// TwinCAT 3 PLC project ToolChanger
// ProgramVersion: 3.1.4023.0
// libraries:
//   CmpBitmapPool, * (System)
//   Tc2_MC2, * (Beckhoff Automation GmbH)
//   Tc2_NC, * (Beckhoff Automation GmbH)
//   Tc2_Standard, * (Beckhoff Automation GmbH)
//   Tc2_System, * (Beckhoff Automation GmbH)
//   Tc2_Utilities, * (Beckhoff Automation GmbH)
//   Tc3_Module, * (Beckhoff Automation GmbH)
//   VisuDialogs, * (System)
//   VisuSymbols,3.5.10.0,System
// project tree:
//   / GlobalTextList.TcGTLO, PlcTask.TcTTO, Visualization Manager.TcVMO (not stored)
//   GVLs/ Allengage.TcGVL, CLEANout.TcGVL, cntrlstate.TcGVL, DSin.TcGVL, DSout.TcGVL, engage.TcGVL, TCin.TcGVL, TCout.TcGVL
//   POUs/FBs/Cleaner/ fb_cleanIn.TcPOU, fb_cleanOut.TcPOU
//   POUs/FBs/Combined/ fb_engageDockAll.TcPOU, fb_engageUndockAll.TcPOU
//   POUs/FBs/DS/ fb_dsopenclose.TcPOU
//   POUs/FBs/Safety/ fb_NozCheck.TcPOU, fb_switchclkcheck.TcPOU
//   POUs/FBs/TC/ fb_dock.TcPOU, fb_toggleVal.TcPOU, fb_undock.TcPOU
//   POUs/FBs/Testing/ fb_testpiston.TcPOU
//   POUs/ MAIN.TcPOU
//   VISUs/ ImagePool.TcIPO (not stored), Visualization.TcVIS
// real-time tasks:
//   TASK PlcTask: cycle T#10ms, priority 20, ADS port 350
// motion (NC):
//   TASK NC-Task 1 SAF: cycle T#2ms, priority 4, ADS port 501
//   TASK NC-Task 1 SVB: cycle T#10ms, priority 8, ADS port 511
//   AXIS Axis 1 (id 1)
//     Velo: SlowManual=20, FastManual=20
//     OtherSettings: AllowMotionCmdToSlave=true
//     encoder EncType=1
//     drive DrvType=5
//       Analog: TorqueSetpointScale=10, ScaleFactorActTorque=0.1
//       TimeComp: TaskDelayCycles=1
//     controller CtrType=1
//       CtrPara: PriorControlFactor=1
//         Observer: BandWidth=20
// I/O:
//   DEVICE Device 1 (EtherCAT), AmsNetId 192.168.1.12.2.1
//     Term 1 (EK1200) [EK1200-5000 EtherCAT Power supply (2A E-Bus)]
//       Term 2 (EL1008) [EL1008 8Ch. Dig. Input 24V, 3ms]
//       Term 3 (EL2008) [EL2008 8Ch. Dig. Output 24V, 0.5A]
//       Term 4 (EK1110) [EK1110 EtherCAT extension]
//   DEVICE Device 4 (COM Port)
// variable links:
//   ToolChanger/ToolChanger Instance <-> Device 1 (EtherCAT)/Term 1 (EK1200)/Term 2 (EL1008)
//     PlcTask Inputs/DSin.endStopBck <-> Channel 5/Input
//     PlcTask Inputs/DSin.endStopFrnt <-> Channel 4/Input
//     PlcTask Inputs/TCin.CollisionSW <-> Channel 2/Input
//     PlcTask Inputs/TCin.ProxDwn <-> Channel 1/Input
//     PlcTask Inputs/TCin.ProxUp <-> Channel 3/Input
//   ToolChanger/ToolChanger Instance <-> Device 1 (EtherCAT)/Term 1 (EK1200)/Term 3 (EL2008)
//     PlcTask Outputs/DSout.servoBackward <-> Channel 4/Output
//     PlcTask Outputs/DSout.servoForward <-> Channel 2/Output
//     PlcTask Outputs/TCout.valvepull <-> Channel 1/Output
//     PlcTask Outputs/TCout.valvepush <-> Channel 3/Output
//   ToolChanger/ToolChanger Instance <-> NC-Task 1 SAF/Axes/Axis 1
//     PlcTask Inputs/MAIN.opcl.ax1.NcToPlc <-> Outputs/ToPlc
//     PlcTask Outputs/MAIN.opcl.ax1.PlcToNc <-> Inputs/FromPlc

CONFIGURATION ToolChanger
    RESOURCE PLC ON TwinCAT3
        TASK PlcTask(INTERVAL := T#10ms, PRIORITY := 20);
        PROGRAM MAIN WITH PlcTask : MAIN;
    END_RESOURCE
END_CONFIGURATION

// ---- GVLs/Allengage.TcGVL
{attribute 'qualified_only'}
VAR_GLOBAL
	cleanInd: BOOL := FALSE;
	cleanOutd: BOOL := FALSE;
	cleanInu: BOOL := FALSE;
	cleanOutu: BOOL := FALSE;
	undock: BOOL := FALSE;
	dock: BOOL := FALSE;
	stepopen: BOOL := FALSE;
	stepclose: BOOL := FALSE;
	stepper : BOOL := FALSE;
END_VAR

// ---- GVLs/CLEANout.TcGVL
{attribute 'qualified_only'}
VAR_GLOBAL
	// Inside cleaner valve
	inValve AT %Q*: BOOL;
	// Outside cleaner valve
	outValve AT %Q*: BOOL;
	
	// ADD COVER SERVO TO SOLUTION
END_VAR

// ---- GVLs/cntrlstate.TcGVL
{attribute 'qualified_only'}
VAR_GLOBAL
	undock: BOOL;
	dock: BOOL;
	cleanin: BOOL;
	cleanout: BOOL;
	piston_moving: BOOL;
	cover_moving: BOOL;
END_VAR

// ---- GVLs/DSin.TcGVL
{attribute 'qualified_only'}
VAR_GLOBAL
	// Cover switch back
	endStopBck AT %I*: BOOL;
	// Cover switch front
	endStopFrnt AT %I*: BOOL;
	// stepper engagement
	open : BOOL := FALSE;
	close : BOOL := FALSE;
	ID: INT;
END_VAR

// ---- GVLs/DSout.TcGVL
{attribute 'qualified_only'}
VAR_GLOBAL
	//ADD COVER SERVO AND STEPPER MOTOR TO SOLUTION
	servoBackward AT %Q*: BOOL := FALSE;
	servoForward AT %Q*: BOOL := false;
END_VAR

// ---- GVLs/engage.TcGVL
{attribute 'qualified_only'}
VAR_GLOBAL
	cleanIn: BOOL := FALSE;
	cleanOut: BOOL := FALSE;
	undock: BOOL := FALSE;
	dock: BOOL := FALSE;
	stepopen: BOOL := FALSE;
	stepclose: BOOL := FALSE;
	stepper : BOOL := FALSE;
	allundock: BOOL :=FALSE;
	alldock: BOOL :=FALSE;
	pisttest : BOOL := FALSE;
END_VAR

// ---- GVLs/TCin.TcGVL
{attribute 'qualified_only'}
VAR_GLOBAL
	// Upper inductive sensor
	ProxUp AT %I*: BOOL;
	// Lower inductive sensor
	ProxDwn AT %I*: BOOL;
	// Safety limit switch
	CollisionSW AT %I*: BOOL;
	// Most significant bit
	ID1 AT %I*: BOOL := TRUE;
	// Middle bit
	ID2 AT %I*: BOOL;
	// Least significant bit
	ID3 AT %I*: BOOL;
	toolOn : BOOL;
END_VAR

// ---- GVLs/TCout.TcGVL
{attribute 'qualified_only'}
VAR_GLOBAL
	// Dual valve control
	valvepush AT %Q*: BOOL := TRUE;
	valvepull AT %Q*: BOOL;
	// Limit switch clock signal
	SwCLK AT %Q*: BOOL;
END_VAR

// ---- POUs/MAIN.TcPOU
PROGRAM MAIN
VAR
	cleanin: fb_cleanIn;
	cleanout: fb_cleanOut;
	undock: fb_undock;
	dock: fb_dock;
	switchclk: fb_switchclkcheck;
	opcl: fb_dsopenclose;
	allundock: fb_engageUndockAll;
	alldock: fb_engageDockAll;
	stop : TC_Stop;
	pisttest: fb_testpiston;
END_VAR

(*always running*)

IF TCin.toolOn THEN
	switchclk();
END_IF

(*engaged manually*)
IF engage.stepper THEN
	opcl();
END_IF

IF engage.cleanIn THEN
	cntrlstate.cleanin := FALSE;
	cleanin(done := cntrlstate.cleanin);
	IF cntrlstate.cleanin THEN
		engage.cleanIn := FALSE;
	END_IF
END_IF

IF engage.cleanOut THEN
	cntrlstate.cleanout := FALSE;
	cleanout(done := cntrlstate.cleanout);
	IF cntrlstate.cleanout THEN
		engage.cleanOut := FALSE;
	END_IF
END_IF

IF engage.undock THEN
	cntrlstate.undock := FALSE;
	undock();
	IF cntrlstate.undock THEN
		engage.undock := FALSE;
	END_IF
END_IF

IF engage.dock THEN
	cntrlstate.dock := FALSE;
	dock(toolID := 4);
	IF cntrlstate.dock THEN
		engage.dock := FALSE;
	END_IF
END_IF


(*engage a sequence*)
IF engage.allundock THEN
	allundock();
END_IF

IF engage.alldock THEN
	alldock();
END_IF

(*errorHandle stopping plc*)
IF NOT switchclk.swXgood THEN
	stop(STOP:=TRUE);
END_IF


(*TESTING*)
IF engage.pisttest THEN
	pisttest();
END_IF

END_PROGRAM

// ---- POUs/FBs/Cleaner/fb_cleanIn.TcPOU
FUNCTION_BLOCK fb_cleanIn
VAR_INPUT
	IN: BOOL;
END_VAR
VAR_OUTPUT
END_VAR
VAR
	wait: TON;
	step: INT;
END_VAR

VAR_IN_OUT
	done: BOOL;
END_VAR

CASE step OF
	0:
		IF NOT done THEN
			cleanout.inValve := TRUE;
			wait(IN := TRUE, PT := T#5S);
			step := 1;
		END_IF
	1:
		IF wait.Q THEN
			wait.IN := FALSE;
			cleanout.inValve := FALSE;
			step := 2;
		END_IF
		
	2: 
		step := 0;
		done := TRUE;
	
END_CASE
wait();

END_FUNCTION_BLOCK

// ---- POUs/FBs/Cleaner/fb_cleanOut.TcPOU
FUNCTION_BLOCK fb_cleanOut
VAR_INPUT
END_VAR
VAR_OUTPUT
END_VAR
VAR
	step: INT;
	wait: TON;
END_VAR

VAR_IN_OUT
	done: BOOL;
END_VAR

CASE step OF
	0:
		IF NOT done THEN
			cleanout.outValve := TRUE;
			wait(IN := TRUE, PT := T#5S);
			step := 1;
		END_IF
	1:
		IF wait.Q THEN
			wait.IN := FALSE;
			cleanout.outValve := FALSE;
			step := 2;
		END_IF
		
	2: 
		step := 0;
		done := TRUE;
	
END_CASE
wait();

END_FUNCTION_BLOCK

// ---- POUs/FBs/TC/fb_undock.TcPOU
FUNCTION_BLOCK fb_undock
VAR_INPUT
END_VAR
VAR_OUTPUT
END_VAR
VAR
	step: INT;
	unLock: fb_toggleVal;
END_VAR

CASE step OF
	0:
		IF NOT tcin.ProxUp THEN
			unLock(IN:= TRUE);
			unLock.IN := FALSE;
			cntrlstate.piston_moving := TRUE;
			step := 1;
		END_IF
	1: 
		IF tcin.ProxUp AND tcin.ProxUp THEN
			 cntrlstate.undock := TRUE;
			 cntrlstate.piston_moving := FALSE;
			 step := 0;
		END_IF
	99:
		//ERROR HANDLING
END_CASE
unLock();
(*
CASE step OF
	0:
		IF tcin.ProxDwn THEN
			unLock(IN:= TRUE);
			unLock.IN := FALSE;
			cntrlstate.piston_moving := TRUE;
			step := 1;
		END_IF
	1: 
		IF tcin.ProxUp AND NOT tcin.ProxDwn THEN
			 cntrlstate.undock := TRUE;
			 cntrlstate.piston_moving := FALSE;
			 step := 0;
		END_IF
	99:
		//ERROR HANDLING
END_CASE
unLock();*)

END_FUNCTION_BLOCK

// ---- POUs/FBs/TC/fb_toggleVal.TcPOU
FUNCTION_BLOCK fb_toggleVal
VAR_INPUT
	IN: BOOL;
END_VAR
VAR_OUTPUT
END_VAR
VAR
END_VAR

IF IN = TRUE AND TCin.ProxUp THEN
	TCout.valvepush := TRUE;
	TCout.valvepull := FALSE;
ELSIF IN = TRUE AND not TCin.ProxUp THEN
	TCout.valvepull := TRUE;
	TCout.valvepush := FALSE;
END_IF

(*
IF IN = TRUE AND TCin.ProxUp THEN
	TCout.valve := FALSE;
ELSIF IN = TRUE AND TCin.ProxDwn THEN
	TCout.valve := TRUE;
END_IF*)

END_FUNCTION_BLOCK

// ---- POUs/FBs/TC/fb_dock.TcPOU
FUNCTION_BLOCK fb_dock
VAR_INPUT
	toolID: int;
END_VAR
VAR_OUTPUT
END_VAR
VAR
	step: INT;
	Lock: fb_toggleVal;
	IDcheck: fb_NozCheck;
END_VAR

CASE step OF
	0:
		IF tcin.ProxUp THEN
			Lock(IN:= TRUE);
			Lock.IN := FALSE;
			cntrlstate.piston_moving := TRUE;
			step := 1;
		END_IF
	1: 
		IF NOT tcin.ProxUp AND NOT tcin.ProxUp THEN
			IDcheck(inID := toolID);
			cntrlstate.piston_moving := FALSE;
			IF IDcheck.good THEN
				cntrlstate.dock := TRUE;
				step := 0;
			ELSIF NOT IDcheck.good THEN
				step := 99;
			END_IF
			
		END_IF
	99:
		//ERROR HANDLING
END_CASE

END_FUNCTION_BLOCK

// ---- POUs/FBs/Safety/fb_NozCheck.TcPOU
FUNCTION_BLOCK fb_NozCheck
VAR_INPUT
	inID: INT;
END_VAR
VAR_OUTPUT
	good: BOOL;
	done: BOOL;
END_VAR
VAR
	outID: INT;
END_VAR

// example (ID1 = 0, ID2 = 1, ID3 = 1)=011 => outID = 3
good := FALSE;
done := FALSE;
IF TCin.ID1 = FALSE AND TCin.ID2 = FALSE AND TCin.ID3 = FALSE THEN
	outID := 0;
ELSIF TCin.ID1 = FALSE AND TCin.ID2 = FALSE AND TCin.ID3 = TRUE THEN
	outID := 1;
ELSIF TCin.ID1 = FALSE AND TCin.ID2 = TRUE AND TCin.ID3 = FALSE THEN
	outID := 2;	
ELSIF TCin.ID1 = FALSE AND TCin.ID2 = TRUE AND TCin.ID3 = TRUE THEN
	outID := 3;
ELSIF TCin.ID1 = TRUE AND TCin.ID2 = FALSE AND TCin.ID3 = FALSE THEN
	outID := 4;
ELSIF TCin.ID1 = TRUE AND TCin.ID2 = FALSE AND TCin.ID3 = TRUE THEN
	outID := 5;	
ELSIF TCin.ID1 = TRUE AND TCin.ID2 = TRUE AND TCin.ID3 = FALSE THEN
	outID := 6;	
ELSIF TCin.ID1 = TRUE AND TCin.ID2 = TRUE AND TCin.ID3 = TRUE THEN
	outID := 7;	
END_IF

IF inID = outID THEN
	good := TRUE;
	done := TRUE;
ELSIF inID <> outID THEN
	good := FALSE;
	done := TRUE;
END_IF

END_FUNCTION_BLOCK

// ---- POUs/FBs/Safety/fb_switchclkcheck.TcPOU
FUNCTION_BLOCK fb_switchclkcheck
VAR_OUTPUT
	swXgood: BOOL := TRUE;
END_VAR
VAR
	prev_clk: BOOL;
END_VAR

(*This function block sends an alternating signal at a frequency of 100 Hz, and checks whether 
it has been altered from previous check*)

(*
TCout.SwCLK := NOT TCout.SwCLK;	
IF prev_clk = TCout.SwCLK THEN
	swXgood := FALSE;
ELSE 
	swXgood := TRUE;
END_IF
prev_clk := TCout.SwCLK; //only for testing => when doing physical setup => prev_clk := TCin.CollisionSW; 
*)

IF TCin.CollisionSW = FALSE THEN
	// STOP
END_IF

END_FUNCTION_BLOCK

// ---- POUs/FBs/DS/fb_dsopenclose.TcPOU
FUNCTION_BLOCK fb_dsopenclose
VAR_INPUT
END_VAR
VAR_OUTPUT
END_VAR
VAR
	ax1: AXIS_REF;
	McJog: MC_Jog;
	McPower: MC_Power;
	McReset: MC_Reset;
	McStop: MC_Stop;
	iState: INT;
END_VAR

(*McPower(Axis := ax1, Enable := TRUE, Enable_Positive := TRUE, Enable_Negative := TRUE);
McReset(Axis := ax1);
McJog(Axis := ax1);
CASE iState OF 
	0: 
		iState := 10;
	
	10:
		McReset(Axis:= ax1, Execute := TRUE);
		IF McReset.Done THEN
			iState := 20;
		ELSIF McReset.Error THEN
			iState := 999;
		END_IF
	
	20:
		IF McPower.Status THEN
			iState := 30;
		END_IF
		
	30:
		IF engage.stepopen OR DSin.open THEN
			cntrlstate.cover_moving := TRUE;
			McJog(Axis := ax1, JogForward := NOT DSin.endStopBck, Velocity := 20);
			IF DSin.endStopBck THEN
				cntrlstate.cover_moving := FALSE;
				engage.stepper := FALSE;
				engage.stepopen := FALSE;
				DSin.open := FALSE;
			END_IF
		ELSIF engage.stepclose OR DSin.close THEN
			cntrlstate.cover_moving := TRUE;
			McJog(Axis := ax1, JogBackwards := NOT DSin.endStopFrnt, Velocity := 20);
			IF DSin.endStopFrnt THEN
				cntrlstate.cover_moving := FALSE;
				engage.stepper := FALSE;
				engage.stepclose := FALSE;
				DSin.close := FALSE;
			END_IF
		END_IF
END_CASE
*)
IF engage.stepopen OR DSin.open THEN
	cntrlstate.cover_moving := TRUE;
	DSout.servoBackward := TRUE;
	IF DSin.endStopBck = FALSE THEN
		DSout.servoBackward := FALSE;
		cntrlstate.cover_moving := FALSE;
		engage.stepper := FALSE;
		engage.stepopen := FALSE;
		DSin.open := FALSE;
	END_IF
ELSIF engage.stepclose OR DSin.close THEN
	cntrlstate.cover_moving := TRUE;
	DSout.servoForward := TRUE;
	IF DSin.endStopFrnt = FALSE THEN
		DSout.servoForward := FALSE;
		cntrlstate.cover_moving := FALSE;
		engage.stepper := FALSE;
		engage.stepclose := FALSE;
		DSin.close := FALSE;
	END_IF
END_IF

END_FUNCTION_BLOCK

// ---- POUs/FBs/Combined/fb_engageUndockAll.TcPOU
FUNCTION_BLOCK fb_engageUndockAll
VAR_INPUT
END_VAR
VAR_OUTPUT
END_VAR
VAR
	step: INT;
	cleanin: fb_cleanIn;
	cleanout: fb_cleanOut;
	undock: fb_undock;
	dock: fb_dock;
	opcl: fb_dsopenclose;
END_VAR

CASE step OF
	0:
		IF Allengage.cleanOutu THEN
			cntrlstate.cleanout := FALSE;
			cleanout(done := cntrlstate.cleanout);
			IF cntrlstate.cleanout THEN
				Allengage.cleanOutu := FALSE;
				Allengage.stepper := TRUE;
				step := 1;
			END_IF
		END_IF
	1: 
		IF Allengage.stepper THEN
			DSin.open := TRUE;
			opcl();
			IF NOT DSin.open THEN
				step := 2;
				Allengage.undock := TRUE;
				Allengage.stepper := FALSE;
			END_IF
		END_IF
	
	2:
		IF Allengage.undock THEN
			cntrlstate.undock := FALSE;
			undock();
			IF cntrlstate.undock THEN
				Allengage.undock := FALSE;
				Allengage.stepper := TRUE;
				step := 3;
			END_IF
		END_IF
	
	3:
		IF Allengage.stepper THEN
			DSin.close := TRUE;
			opcl();
			IF NOT DSin.close THEN
				step := 4;
				Allengage.stepper := FALSE;
			END_IF
		END_IF
		
	4:
		engage.allundock := FALSE;
		step := 0;
END_CASE

END_FUNCTION_BLOCK

// ---- POUs/FBs/Combined/fb_engageDockAll.TcPOU
FUNCTION_BLOCK fb_engageDockAll
VAR_INPUT
END_VAR
VAR_OUTPUT
END_VAR
VAR
	cleanin: fb_cleanIn;
	cleanout: fb_cleanOut;
	step: INT;
	clop: fb_dsopenclose;
	dock: fb_dock;
END_VAR

CASE step OF
	0:
		IF Allengage.cleanOutd THEN
			cntrlstate.cleanout := FALSE;
			cleanout(done := cntrlstate.cleanout);
			IF cntrlstate.cleanout THEN
				Allengage.cleanOutd := FALSE;
				Allengage.cleanInd := TRUE;
				step := 1;
			END_IF
		END_IF
		
	1:
		IF Allengage.cleanInd THEN
			cntrlstate.cleanin := FALSE;
			cleanin(done := cntrlstate.cleanin);
			IF cntrlstate.cleanin THEN
				Allengage.cleanInd := FALSE;
				Allengage.stepper := TRUE;
				step := 2;
			END_IF
		END_IF
		
	2: 
		IF Allengage.stepper THEN
			DSin.open := TRUE;
			clop();
			IF NOT DSin.open THEN
				step := 3;
				Allengage.dock := TRUE;
				Allengage.stepper := FALSE;
			END_IF
		END_IF
	
	3:
		IF Allengage.dock THEN
			cntrlstate.dock := FALSE;
			dock(toolID := DSin.ID);
			IF cntrlstate.dock THEN
				Allengage.dock := FALSE;
				Allengage.stepper := TRUE;
				step := 4;
			END_IF
		END_IF
	
	4:
		IF Allengage.stepper THEN
			DSin.close := TRUE;
			clop();
			IF NOT DSin.close THEN
				step := 5;
				Allengage.stepper := FALSE;
			END_IF
		END_IF
		
	5:
		engage.alldock := FALSE;
		step := 0;
END_CASE

END_FUNCTION_BLOCK

// ---- POUs/FBs/Testing/fb_testpiston.TcPOU
FUNCTION_BLOCK fb_testpiston
VAR_INPUT
END_VAR
VAR_OUTPUT
END_VAR
VAR
	step: INT;
	wait1: TON;
	wait2: TON;
	unlock: INT;
	failUp: INT;
	failDown: INT;
	lock: INT;
	wait: INT;
	totalFail: INT;
	wait3: TON;
	wait4: TON;
END_VAR

IF (unlock > 50 AND lock > 50) OR totalFail <> 0 THEN
	ADSLOGDINT( msgCtrlMask := ADSLOG_MSGTYPE_HINT OR ADSLOG_MSGTYPE_MSGBOX, 
                    msgFmtStr := 'test Msg: Test DONE! Number of fails: %d', dintArg:= totalFail);
	ADSLOGDINT( msgCtrlMask := ADSLOG_MSGTYPE_HINT OR ADSLOG_MSGTYPE_MSGBOX, 
                    msgFmtStr := '%d Unlock fails', dintArg:= failUp);
	ADSLOGDINT( msgCtrlMask := ADSLOG_MSGTYPE_HINT OR ADSLOG_MSGTYPE_MSGBOX, 
                    msgFmtStr := '%d Lock fails', dintArg:= failDown);
	wait1.IN := FALSE;
	wait2.IN := FALSE;
	unlock := 0;
	lock := 0;
	totalFail := 0;
	failDown := 0;
	failUp := 0;
	step := 1000;
END_IF

CASE step OF
	0: 
		step := 10;
	10:
		wait3(IN := TRUE, PT := T#1000MS);
		IF tcin.ProxUp THEN
			IF wait3.Q THEN
				wait2.IN := FALSE;
				wait3.IN := FALSE;
				tcout.valvePush := TRUE;
				tcout.valvePull := FALSE;
				wait1(IN := TRUE, PT := T#10S);
				step := 20;
				unlock := unlock + 1;
			END_IF
		ELSIF wait2.Q THEN
			step := 991;
		END_IF
		
	20:
		wait4(IN := TRUE, PT := T#1000MS);
		IF tcin.ProxDwn THEN
			IF wait4.Q THEN
				wait4.IN := FALSE;
				wait1.IN := FALSE;
				tcout.valvePull := TRUE;
				tcout.valvePush := FALSE;
				wait2(IN := TRUE, PT := T#10S);
				step := 10;
				lock := lock + 1;
			END_IF
		ELSIF wait1.Q THEN
			step := 992;
		END_IF
		
	991:
		failUp := failUp + 1;
		step := 999;
		
	992:
		failDown := failDown + 1;
		step := 999;
		
	999:
		totalFail := totalFail + 1;
		wait1.IN := FALSE;
		wait2.IN := FALSE;
		step := 1001;
	
	1000:
		step := 0;
		
	1001:
		
END_CASE
wait4();
wait3();
wait2();
wait1();

END_FUNCTION_BLOCK

// ---- GlobalTextList.TcGTLO
TEXTLIST GlobalTextList
  736 = 'Activate'
  606 = 'Clean Inside'
  691 = 'Clean Outside'
  249 = 'Cleaning station'
  84 = 'Close Docking Station Cover'
  649 = 'Dock Sequence'
  364 = 'Docking'
  545 = 'Docking Maneuvers'
  151 = 'Docking Station'
  146 = 'Inductive sensors'
  175 = 'Inductive Sensors'
  731 = 'Manual Control'
  625 = 'Nozzle ID'
  685 = 'Open Docking Station Cover'
  631 = 'Safety'
  374 = 'Safety Switch'
  608 = 'Start'
  734 = 'Tool Changer'
  582 = 'Undock Sequence'
  367 = 'Undocking'
  709 = 'Valves'
END_TEXTLIST

// ---- VISUs/Visualization.TcVIS
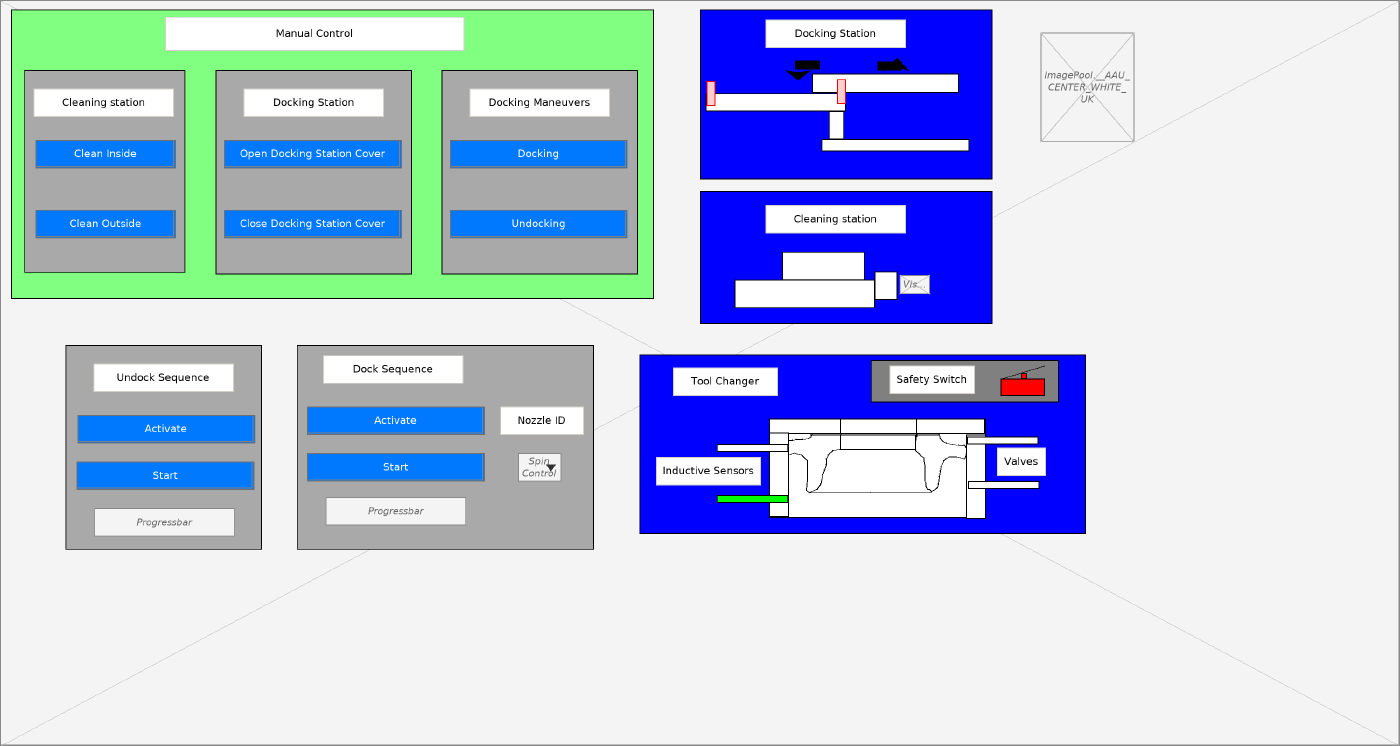
VISUALIZATION Visualization  // 1500x800
    Image (0,0 1500x800), image: ImagePool.Lasercut
    RoundedRectangle (685,380 478x192)
    RoundedRectangle (750,205 313x142)
    RoundedRectangle (750,10 313x182)
    RoundedRectangle (12,10 688x310)
    RoundedRectangle (231,75 210x219)
    RoundedRectangle (26,75 172x217)
    Button (38,150 150x30), "Clean Inside", colour toggle: CLEANout.inValve
        OnMouseClick: toggle engage.cleanIn
    Button (38,225 150x30), "Clean Outside", colour toggle: CLEANout.outValve
        OnMouseClick: toggle engage.cleanOut
    Button (240,150 190x30), "Open Docking Station Cover", colour toggle: engage.stepopen
        OnMouseClick: toggle engage.stepopen
        OnMouseClick: toggle engage.stepper
    Button (240,225 190x30), "Close Docking Station Cover", colour toggle: engage.stepclose
        OnMouseClick: toggle engage.stepclose
        OnMouseClick: toggle engage.stepper
    Textfield (36,95 150x30), "Cleaning station"
    Textfield (261,95 150x30), "Docking Station"
    RoundedRectangle (473,75 210x219)
    Button (482,150 190x30), "Docking", colour toggle: engage.dock
        OnMouseClick: toggle engage.dock
    Button (482,225 190x30), "Undocking", colour toggle: engage.undock
        OnMouseClick: toggle engage.undock
    Textfield (503,95 150x30), "Docking Maneuvers"
    RoundedRectangle (70,370 210x219)
    Button (83,445 190x30), "Activate", colour toggle: engage.allundock
        OnMouseClick: toggle engage.allundock
    Button (82,495 190x30), "Start", colour toggle: Allengage.cleanOutu
        OnMouseClick: toggle Allengage.cleanOutu
    Textfield (100,390 150x30), "Undock Sequence"
    Progressbar (101,545 150x30), variable: MAIN.allundock.step
    Textfield (177,18 320x36), "Manual Control"
    Rectangle (870,79 157x20), colour toggle: cntrlstate.cover_moving
    Rectangle (756,100 150x19)
    Rectangle (888,119 16x30)
    Rectangle (880,149 158x13)
    Textfield (820,21 150x30), "Docking Station"
    Rectangle (787,300 150x30)
    RoundedRectangle (838,270 88x30), colour toggle: cleanout.inValve
    Rectangle (937,291 24x30), colour toggle: cleanout.outValve
    Image (964,295 32x20), colour toggle: cleanout.outValve, image: VisuSymbols.Symbols.ArrowBoldRight
    Textfield (820,220 150x30), "Cleaning station"
    Rectangle (824,449 232x106)
    Rectangle (824,449 231x16)
    Group (843,465 193x63), colour toggle: cntrlstate.piston_moving
        Polyline (25,1) (58,1) (57,17) (49,18) (44,23) (42,27) (42,33) (40,39) (38,44) (36,54) (32,60) (24,63) (21,61) (22,49) (22,37) (22,29) (16,23) (11,22) (8,21) (2,23) (0,15) (2,7) (6,7) (10,6) (17,6) (23,5) (26,3) (27,0)
        Polyline (135,1) (163,1) (164,5) (167,8) (171,10) (184,12) (190,12) (193,17) (192,22) (190,27) (182,25) (174,25) (170,27) (168,29) (165,35) (164,40) (163,46) (162,54) (161,58) (160,59) (157,61) (155,62) (153,60) (151,60) (149,57) (149,53) (148,51) (148,47) (148,43) (148,38) (148,37) (148,34) (147,29)
        Polyline (147,30) (147,26) (144,24) (142,22) (138,18) (138,10) (139,0) (139,3)
        Rectangle (57,1 81x16)
        Line (24,63) (155,62)
    Rectangle (824,464 21x90)
    Rectangle (1035,466 21x90)
    Rectangle (768,476 76x8), colour toggle: TCin.ProxUp
    Rectangle (768,531 76x8), colour toggle: TCin.ProxUp
    Textfield (703,490 112x30), "Inductive Sensors"
    Rectangle (757,87 9x26), colour toggle: DSin.endStopBck
    Rectangle (897,85 9x26), colour toggle: DSin.endStopFrnt
    Textfield (721,394 112x30), "Tool Changer"
    Rectangle (1036,468 76x8), colour toggle: TCout.valvepush
    Rectangle (1037,516 76x8), colour toggle: TCout.valvepull
    Textfield (1068,480 52x30), "Valves"
    RoundedRectangle (318,370 318x219)
    Button (329,436 190x30), "Activate", colour toggle: engage.alldock
        OnMouseClick: toggle engage.alldock
    Button (329,486 190x30), "Start", colour toggle: Allengage.cleanOutd
        OnMouseClick: toggle Allengage.cleanOutd
    Textfield (346,381 150x30), "Dock Sequence"
    Progressbar (349,533 150x30), variable: MAIN.alldock.step
    SpinControl (555,486 46x30), variable: DSin.ID
        tap DSin.ID
    Textfield (536,436 89x30), "Nozzle ID"
    RoundedRectangle (933,386 201x45)
    Rectangle (1072,406 47x18), colour toggle: TCin.CollisionSW
    RoundedRectangle (1094,400 6x6), colour toggle: MAIN.switchclk.swXgood
    Line (1073,406) (1119,392)
    Textfield (953,392 91x30), "Safety Switch"
    Rectangle (940,66 26x9), colour toggle: engage.stepclose
    Polygon (946,76) (961,62) (974,76) (962,72) (956,72), colour toggle: engage.stepclose
    Rectangle (852,65 26x9), colour toggle: engage.stepopen
    Polygon (841,75) (855,86) (869,75) (857,77) (855,77), colour toggle: engage.stepopen
    Rectangle (900,449 82x16)
    Image (1115,35 100x117), image: ImagePool.__AAU_CENTER_WHITE_UK
END_VISUALIZATION
